// TIA Portal project "学习代码" (V15.1)

(* hardware
DEVICE "S7-1200 station_1"  S7-1200 Station
   slot 0: "Rack_0"  S7-1200 Rack  Rack  V1.0
   slot 1: "PLC_1"  CPU 1214C DC/DC/DC  6ES7 214-1AG40-0XB0  V4.2
   slot 2: "AQ 4x14BIT_1"  6ES7 232-4HD32-0XB0  V2.0
   slot 101: "CM 1241 (RS232)_1"  6ES7 241-1AH32-0XB0  V2.2
*)

// ===== PLC "PLC_1"  CPU 1214C DC/DC/DC =====

VAR_GLOBAL   // PLC tag table "默认变量表"
   "点动模式状态指示灯" AT %Q0.0 : Bool;
   "点动模式标志位" AT %M100.2 : Bool;
   "Last_Status_2" AT %M100.1 : Bool;
   "Last_Status_1" AT %M100.0 : Bool;
   "启动" AT %I1.0 : Bool;
   "停止" AT %I1.1 : Bool;
   "运行标志位" AT %M10.0 : Bool;
   "测试" AT %I1.2 : Bool;
   "测试运行标志位" AT %M10.1 : Bool;
   "传送带运行" AT %Q1.0 : Bool;
   "点动正运行标志位" AT %M10.2 : Bool;
   "点动正" AT %I2.0 : Bool;
   "点动负" AT %I2.1 : Bool;
   "点动负运行标志位" AT %M10.3 : Bool;
   "点动模式选择按钮" AT %I0.0 : Bool;
   "TP输入" AT %I3.0 : Bool;
   "TP输出" AT %Q3.0 : Bool;
   "TON输入" AT %I3.1 : Bool;
   "TON输出" AT %Q3.1 : Bool;
   "TOF输入" AT %I3.2 : Bool;
   "TOF输出" AT %Q3.2 : Bool;
   "TONR输入" AT %I3.3 : Bool;
   "TONR输出" AT %Q3.3 : Bool;
   "TONR复位" AT %I3.4 : Bool;
   "CTU输入" AT %I4.0 : Bool;
   "CTU输出" AT %Q4.0 : Bool;
   "CTD输入" AT %I4.1 : Bool;
   "CTD输出" AT %Q4.1 : Bool;
   "CTUD输入增加" AT %I4.2 : Bool;
   "CTUD输出" AT %Q4.2 : Bool;
   "CTUD输入减少" AT %I4.3 : Bool;
   "比较指令输出" AT %Q4.3 : Bool;
   "数学函数输入" AT %I4.4 : Bool;
   "Clock_1Hz" AT %I4.5 : Bool;
   "Last_Status" AT %M50.0 : Bool;
   "电机1启动信号" AT %I5.0 : Bool;
   "电机1停止信号" AT %I5.1 : Bool;
   "电机1频率加信号" AT %I5.2 : Bool;
   "电机1频率减信号" AT %I5.3 : Bool;
   "电机1运行" AT %Q5.0 : Bool;
   "电机1运行指示灯" AT %Q5.1 : Bool;
   "AQ1" AT %QW96 : Int;
   "System_Byte" AT %MB1 : Byte;
   "FirstScan" AT %M1.0 : Bool;
   "DiagStatusUpdate" AT %M1.1 : Bool;
   "AlwaysTRUE" AT %M1.2 : Bool;
   "AlwaysFALSE" AT %M1.3 : Bool;
END_VAR

TYPE "电机启停运行及速度控制_数据类型"
   STRUCT
      设定运行时间 : Time;
      运行标志 : Bool;
      运行时间到 : Bool;
      频率加信号上次状态 : Bool;
      频率减信号上次状态 : Bool;
      TON_DB : IEC_TIMER;
      给定频率 : Real;
   END_STRUCT;
END_TYPE

DATA_BLOCK "Counter_Data"   // DB1
{ S7_Optimized_Access := 'TRUE' }
VERSION : 0.1
   VAR RETAIN
      CTU : IEC_COUNTER;
   END_VAR
   VAR
      Static_2 : Array[0..1] of IEC_COUNTER;
   END_VAR
BEGIN
END_DATA_BLOCK

DATA_BLOCK "比较指令DB"   // DB2
{ S7_Optimized_Access := 'TRUE' }
VERSION : 0.1
   VAR
      不等于 : Array[0..1] of Int;
      大于 : Real;
      小于 : Time;
      小于等于 : Time_Of_Day;
      大于等于 : DTL;
      INRANGE : Int;
      OUTRANGE : Int;
   END_VAR
BEGIN
END_DATA_BLOCK

DATA_BLOCK "Time_Data"   // DB3
{ S7_Optimized_Access := 'TRUE' }
VERSION : 0.1
   VAR
      TP_DB : IEC_TIMER;
      TON_DB : IEC_TIMER;
      Timer_DB : Array[0..1] of IEC_TIMER;
   END_VAR
BEGIN
END_DATA_BLOCK

DATA_BLOCK "数学函数DB"   // DB4
{ S7_Optimized_Access := 'TRUE' }
VERSION : 0.1
   VAR
      Data1 : Array[0..3] of Int;
      Data2 : Array[0..3] of Int;
      Data3 : Array[0..3] of Real;
      Data4 : Array[0..3] of DInt;
      Data5 : Array[0..1] of DInt;
      Data6 : Array[0..4] of Int;
      Data7 : Array[0..5] of Int;
   END_VAR
BEGIN
END_DATA_BLOCK

DATA_BLOCK "电机启停运行及速度控制_DB"   // DB5
{ S7_Optimized_Access := 'TRUE' }
VERSION : 0.1
   VAR
      电机 : Array[1..4] of "电机启停运行及速度控制_数据类型";
   END_VAR
BEGIN
END_DATA_BLOCK

DATA_BLOCK "电机启停运行及速度控制_FB_DB"   // DB6
{ S7_Optimized_Access := 'TRUE' }
VERSION : 0.1
// stored: InstanceOfName 电机启停运行及速度控制_FB
"电机启停运行及速度控制_FB"
BEGIN
END_DATA_BLOCK

DATA_BLOCK "MODBUS通讯_DB"   // DB7
{ S7_Optimized_Access := 'FALSE' }
VERSION : 0.1
// stored: InstanceOfName MODBUS通讯
"MODBUS通讯"
BEGIN
END_DATA_BLOCK

FUNCTION_BLOCK "Timer_FB"   // FB1, LAD
{ S7_Optimized_Access := 'TRUE' }
VERSION : 0.1
   VAR
      IEC_Timer_0_Instance : TONR_TIME;
   END_VAR
BEGIN

REGION Network 1
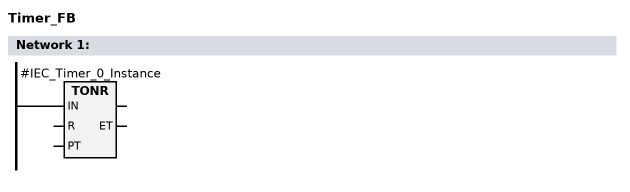
   #IEC_Timer_0_Instance(IN := TRUE);   // TONR
END_REGION
END_FUNCTION_BLOCK

FUNCTION_BLOCK "电机启停运行及速度控制_FB"   // FB2, LAD
{ S7_Optimized_Access := 'TRUE' }
VERSION : 0.1
   VAR_INPUT
      电机启动 : Bool;
      电机停止 : Bool;
      设定运行时间 : Time;
      频率加 : Bool;
      频率减 : Bool;
   END_VAR
   VAR_OUTPUT
      电机输出运行 : Bool;
      运行指示灯 : Bool;
   END_VAR
   VAR_IN_OUT
      给定频率 : Real;
      输出数字量 : Int;
   END_VAR
   VAR
      运行标志 : Bool;
      运行时间到 : Bool;
      IEC_Timer_0_Instance : TON_TIME;
      频率加信号上次状态 : Bool;
      频率减信号上次状态 : Bool;
   END_VAR
   VAR_TEMP
      标定值 : Real;
   END_VAR
   VAR_TEMP   // added for the SCL form of the ladder/FBD networks
      _w1 : Bool;
   END_VAR
BEGIN

REGION Network 1: 启动
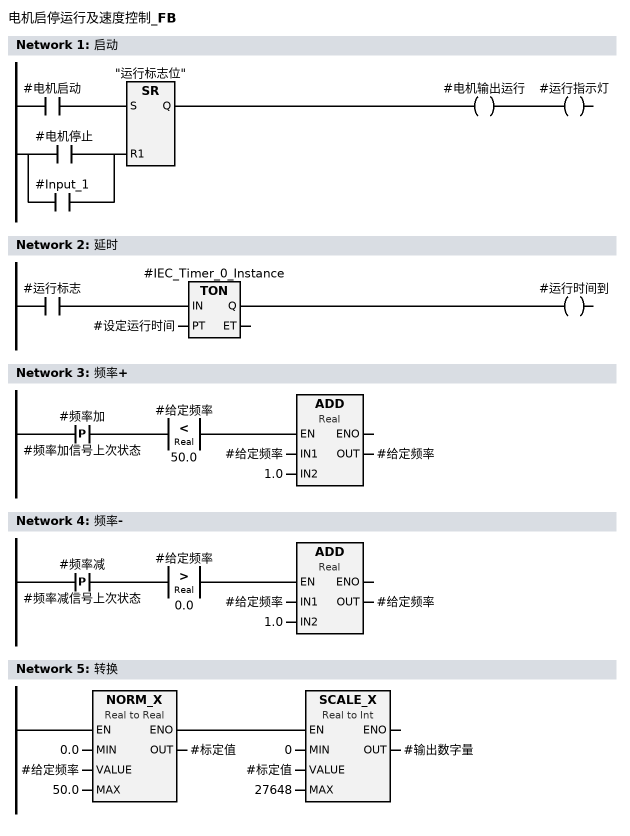
   RUNG wire#powerrail
      Contact( #电机启动 )
      S_SR(operand := "运行标志位", r1 := wire#w1)
      Coil( #电机输出运行 )
      Coil( #运行指示灯 )
   END_RUNG
   RUNG wire#powerrail
      Contact( #电机停止 )
   END_RUNG wire#w1
   RUNG wire#powerrail
      Contact( #Input_1 )
   END_RUNG wire#w1
   // the same network as SCL:
   IF #电机启动 THEN
       "运行标志位" := TRUE;   // SR flip-flop
   END_IF;
   IF #电机停止 OR #Input_1 THEN "运行标志位" := FALSE; END_IF;
   #电机输出运行 := "运行标志位";
   #运行指示灯 := "运行标志位";
END_REGION

REGION Network 2: 延时
   #IEC_Timer_0_Instance(IN := #运行标志, PT := #设定运行时间);   // TON
   #运行时间到 := #IEC_Timer_0_Instance.Q;
END_REGION

REGION Network 3: 频率+
   RUNG wire#powerrail
      P_Contact(operand := #频率加, bit := #频率加信号上次状态)
      { S7_Templates := "SrcType := Real" } LT_Contact(in1 := #给定频率, in2 := 50.0)
      { S7_Templates := "SrcType := Real"; S7_GenerateENO := "TRUE" } Add(in1 := #给定频率, in2 := 1.0, out => #给定频率)
   END_RUNG
   // the same network as SCL:
   #_w1 := #频率加 AND NOT #频率加信号上次状态;   // rising edge of #频率加
   #频率加信号上次状态 := #频率加;
   IF #_w1 AND (#给定频率 < 50.0) THEN #给定频率 := #给定频率 + 1.0; END_IF;
END_REGION

REGION Network 4: 频率-
   RUNG wire#powerrail
      P_Contact(operand := #频率减, bit := #频率减信号上次状态)
      { S7_Templates := "SrcType := Real" } GT_Contact(in1 := #给定频率, in2 := 0.0)
      { S7_Templates := "SrcType := Real"; S7_GenerateENO := "TRUE" } Add(in1 := #给定频率, in2 := 1.0, out => #给定频率)
   END_RUNG
   // the same network as SCL:
   #_w1 := #频率减 AND NOT #频率减信号上次状态;   // rising edge of #频率减
   #频率减信号上次状态 := #频率减;
   IF #_w1 AND (#给定频率 > 0.0) THEN #给定频率 := #给定频率 + 1.0; END_IF;
END_REGION

REGION Network 5: 转换
   RUNG wire#powerrail
      { S7_Templates := "[SrcType := Real, DestType := Real]"; S7_GenerateENO := "TRUE" } Normalize(min := 0.0, value := #给定频率, max := 50.0, out => #标定值)
      { S7_Templates := "[SrcType := Real, DestType := Int]"; S7_GenerateENO := "TRUE" } Scale(min := 0, value := #标定值, max := 27648, out => #输出数字量)
   END_RUNG
   // the same network as SCL:
   // ENO of a box is taken as its EN; it also drops when the box reports an error
   #标定值 := NORM_X(MIN := 0.0, VALUE := #给定频率, MAX := 50.0);
   #输出数字量 := SCALE_X(MIN := 0, VALUE := #标定值, MAX := 27648);
END_REGION
END_FUNCTION_BLOCK

FUNCTION_BLOCK "MODBUS通讯"   // FB3, LAD
{ S7_Optimized_Access := 'FALSE' }
VERSION : 0.1
   VAR_INPUT
      初始化 : Bool;
      正转 : Bool;
      反转 : Bool;
      停止 : Bool;
      频率设定 : Real;
   END_VAR
   VAR_OUTPUT
      输出频率 : Real;
      输出电流 : Real;
      输出电压 : Real;
   END_VAR
   VAR
      Modbus_Comm_Load_DB : Modbus_Comm_Load;
      MB_Com_load : Struct
         Done : Bool;
         Error : Bool;
         Status : Word;
      END_STRUCT;
      MB_Mast_step : USInt;
      Modbus_Master_DB : Modbus_Master;
      MD_Master_write : Struct
         Data_ptr : Array[0..1] of Int;
         Done : Bool;
         Busy : Bool;
         Error : Bool;
         Status : Word;
      END_STRUCT;
      MD_Master_status : Struct
         Data_ptr : Array[0..0] of Int;
         Done : Bool;
         Busy : Bool;
         Error : Bool;
         Status : Word;
      END_STRUCT;
      MD_Master_RD : Struct
         Data_ptr : Array[0..3] of Int;
         Done : Bool;
         Busy : Bool;
         Error : Bool;
         Status : Word;
      END_STRUCT;
   END_VAR
   VAR_TEMP
      设定频率_Real : Real;
      输出频率_Real : Real;
      输出电流_Real : Real;
      输出电压_Real : Real;
   END_VAR
BEGIN

REGION Network 1
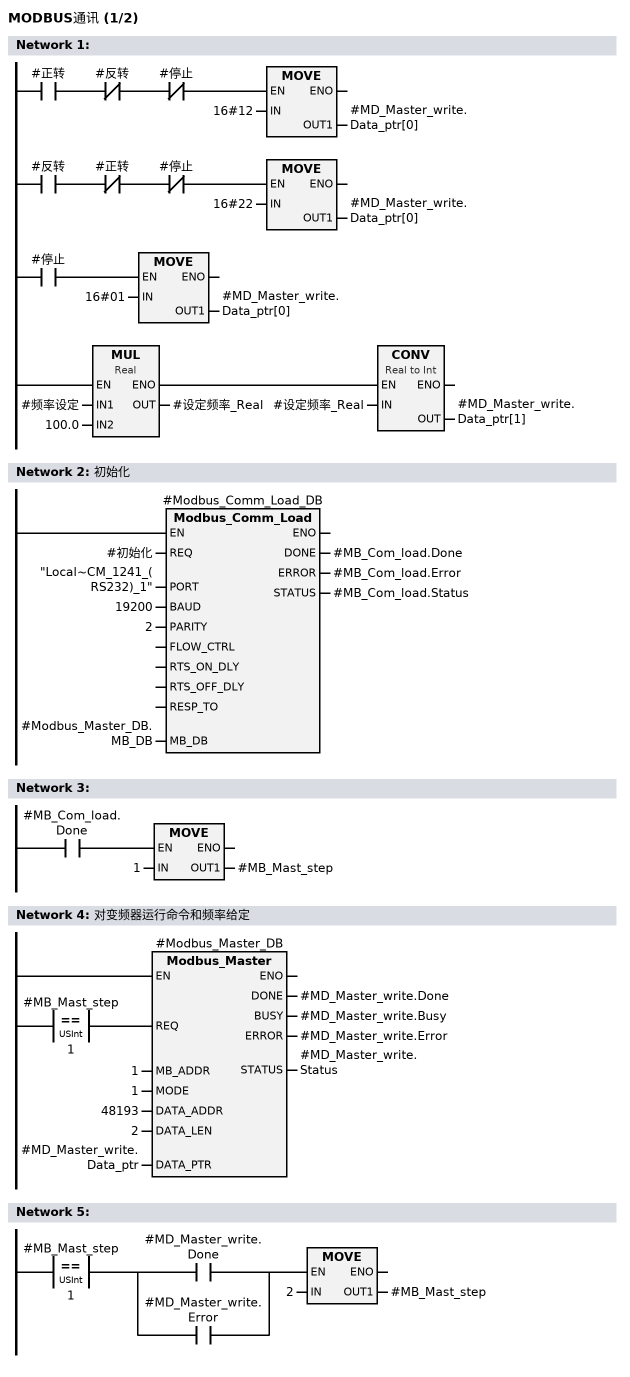
   RUNG wire#powerrail
      Contact( #正转 )
      I_Contact( #反转 )
      I_Contact( #停止 )
      { S7_GenerateENO := "TRUE" } Move(in := 16#12, out1 => #MD_Master_write.Data_ptr[0])
   END_RUNG
   RUNG wire#powerrail
      Contact( #反转 )
      I_Contact( #正转 )
      I_Contact( #停止 )
      { S7_GenerateENO := "TRUE" } Move(in := 16#22, out1 => #MD_Master_write.Data_ptr[0])
   END_RUNG
   RUNG wire#powerrail
      Contact( #停止 )
      { S7_GenerateENO := "TRUE" } Move(in := 16#01, out1 => #MD_Master_write.Data_ptr[0])
   END_RUNG
   RUNG wire#powerrail
      { S7_Templates := "SrcType := Real"; S7_GenerateENO := "TRUE" } Mul(in1 := #频率设定, in2 := 100.0, out => #设定频率_Real)
      { S7_Templates := "[SrcType := Real, DestType := Int]"; S7_GenerateENO := "TRUE" } Convert(in := #设定频率_Real, out => #MD_Master_write.Data_ptr[1])
   END_RUNG
   RUNG wire#powerrail
   END_RUNG
   // the same network as SCL:
   // ENO of a box is taken as its EN; it also drops when the box reports an error
   IF #正转 AND NOT #反转 AND NOT #停止 THEN #MD_Master_write.Data_ptr[0] := 16#12; END_IF;
   IF #反转 AND NOT #正转 AND NOT #停止 THEN #MD_Master_write.Data_ptr[0] := 16#22; END_IF;
   IF #停止 THEN #MD_Master_write.Data_ptr[0] := 16#01; END_IF;
   #设定频率_Real := #频率设定 * 100.0;
   #MD_Master_write.Data_ptr[1] := REAL_TO_INT(#设定频率_Real);
END_REGION

REGION Network 2: 初始化
   #Modbus_Comm_Load_DB(REQ := #初始化,   // Modbus_Comm_Load
                        PORT := "Local~CM_1241_(RS232)_1",
                        BAUD := 19200,
                        PARITY := 2,
                        MB_DB := #Modbus_Master_DB.MB_DB,
                        DONE => #MB_Com_load.Done,
                        ERROR => #MB_Com_load.Error,
                        STATUS => #MB_Com_load.Status);
END_REGION

REGION Network 3
   RUNG wire#powerrail
      Contact( #MB_Com_load.Done )
      { S7_GenerateENO := "TRUE" } Move(in := 1, out1 => #MB_Mast_step)
   END_RUNG
   // the same network as SCL:
   IF #MB_Com_load.Done THEN #MB_Mast_step := 1; END_IF;
END_REGION

REGION Network 4: 对变频器运行命令和频率给定
   #Modbus_Master_DB(REQ := #MB_Mast_step = 1,   // Modbus_Master
                     MB_ADDR := 1,
                     MODE := 1,
                     DATA_ADDR := 48193,
                     DATA_LEN := 2,
                     DATA_PTR := #MD_Master_write.Data_ptr,
                     DONE => #MD_Master_write.Done,
                     BUSY => #MD_Master_write.Busy,
                     ERROR => #MD_Master_write.Error,
                     STATUS => #MD_Master_write.Status);
END_REGION

REGION Network 5
   RUNG wire#powerrail
      { S7_Templates := "SrcType := USInt" } EQ_Contact(in1 := #MB_Mast_step, in2 := 1)
      wire#w1
      Contact( #MD_Master_write.Done )
      wire#w2
      { S7_GenerateENO := "TRUE" } Move(in := 2, out1 => #MB_Mast_step)
   END_RUNG
   RUNG wire#w1
      Contact( #MD_Master_write.Error )
   END_RUNG wire#w2
   // the same network as SCL:
   IF (#MB_Mast_step = 1) AND (#MD_Master_write.Done OR #MD_Master_write.Error) THEN
       #MB_Mast_step := 2;
   END_IF;
END_REGION

REGION Network 6: 读变频器状态
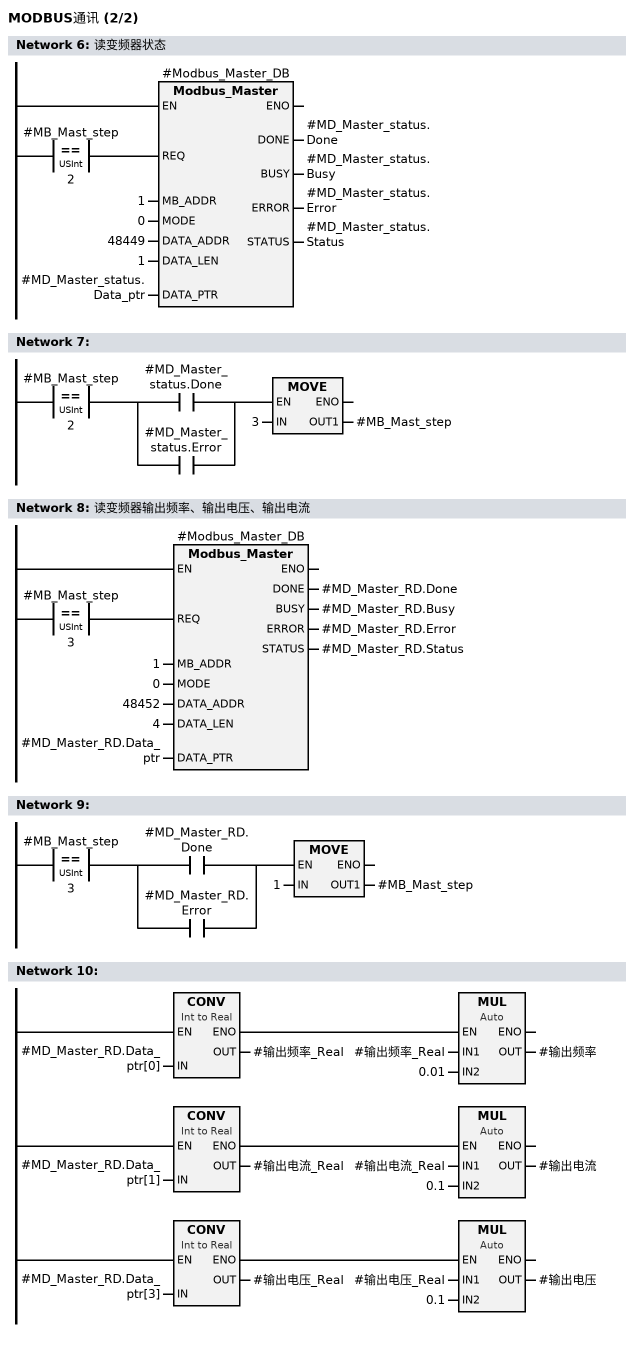
   #Modbus_Master_DB(REQ := #MB_Mast_step = 2,   // Modbus_Master
                     MB_ADDR := 1,
                     MODE := 0,
                     DATA_ADDR := 48449,
                     DATA_LEN := 1,
                     DATA_PTR := #MD_Master_status.Data_ptr,
                     DONE => #MD_Master_status.Done,
                     BUSY => #MD_Master_status.Busy,
                     ERROR => #MD_Master_status.Error,
                     STATUS => #MD_Master_status.Status);
END_REGION

REGION Network 7
   RUNG wire#powerrail
      { S7_Templates := "SrcType := USInt" } EQ_Contact(in1 := #MB_Mast_step, in2 := 2)
      wire#w1
      Contact( #MD_Master_status.Done )
      wire#w2
      { S7_GenerateENO := "TRUE" } Move(in := 3, out1 => #MB_Mast_step)
   END_RUNG
   RUNG wire#w1
      Contact( #MD_Master_status.Error )
   END_RUNG wire#w2
   // the same network as SCL:
   IF (#MB_Mast_step = 2) AND (#MD_Master_status.Done OR #MD_Master_status.Error) THEN
       #MB_Mast_step := 3;
   END_IF;
END_REGION

REGION Network 8: 读变频器输出频率、输出电压、输出电流
   #Modbus_Master_DB(REQ := #MB_Mast_step = 3,   // Modbus_Master
                     MB_ADDR := 1,
                     MODE := 0,
                     DATA_ADDR := 48452,
                     DATA_LEN := 4,
                     DATA_PTR := #MD_Master_RD.Data_ptr,
                     DONE => #MD_Master_RD.Done,
                     BUSY => #MD_Master_RD.Busy,
                     ERROR => #MD_Master_RD.Error,
                     STATUS => #MD_Master_RD.Status);
END_REGION

REGION Network 9
   RUNG wire#powerrail
      { S7_Templates := "SrcType := USInt" } EQ_Contact(in1 := #MB_Mast_step, in2 := 3)
      wire#w1
      Contact( #MD_Master_RD.Done )
      wire#w2
      { S7_GenerateENO := "TRUE" } Move(in := 1, out1 => #MB_Mast_step)
   END_RUNG
   RUNG wire#w1
      Contact( #MD_Master_RD.Error )
   END_RUNG wire#w2
   // the same network as SCL:
   IF (#MB_Mast_step = 3) AND (#MD_Master_RD.Done OR #MD_Master_RD.Error) THEN #MB_Mast_step := 1; END_IF;
END_REGION

REGION Network 10
   RUNG wire#powerrail
      { S7_Templates := "[SrcType := Int, DestType := Real]"; S7_GenerateENO := "TRUE" } Convert(in := #MD_Master_RD.Data_ptr[0], out => #输出频率_Real)
      { S7_GenerateENO := "TRUE" } Mul(in1 := #输出频率_Real, in2 := 0.01, out => #输出频率)
   END_RUNG
   RUNG wire#powerrail
      { S7_Templates := "[SrcType := Int, DestType := Real]"; S7_GenerateENO := "TRUE" } Convert(in := #MD_Master_RD.Data_ptr[1], out => #输出电流_Real)
      { S7_GenerateENO := "TRUE" } Mul(in1 := #输出电流_Real, in2 := 0.1, out => #输出电流)
   END_RUNG
   RUNG wire#powerrail
      { S7_Templates := "[SrcType := Int, DestType := Real]"; S7_GenerateENO := "TRUE" } Convert(in := #MD_Master_RD.Data_ptr[3], out => #输出电压_Real)
      { S7_GenerateENO := "TRUE" } Mul(in1 := #输出电压_Real, in2 := 0.1, out => #输出电压)
   END_RUNG
   // the same network as SCL:
   // ENO of a box is taken as its EN; it also drops when the box reports an error
   #输出频率_Real := INT_TO_REAL(#MD_Master_RD.Data_ptr[0]);
   #输出频率 := #输出频率_Real * 0.01;
   #输出电流_Real := INT_TO_REAL(#MD_Master_RD.Data_ptr[1]);
   #输出电流 := #输出电流_Real * 0.1;
   #输出电压_Real := INT_TO_REAL(#MD_Master_RD.Data_ptr[3]);
   #输出电压 := #输出电压_Real * 0.1;
END_REGION
END_FUNCTION_BLOCK

FUNCTION "传送带控制" : Void   // FC1, LAD
{ S7_Optimized_Access := 'TRUE' }
VERSION : 0.1
   VAR_TEMP   // added for the SCL form of the ladder/FBD networks
      _w1 : Bool;
      _w2 : Bool;
   END_VAR
BEGIN

REGION Network 1
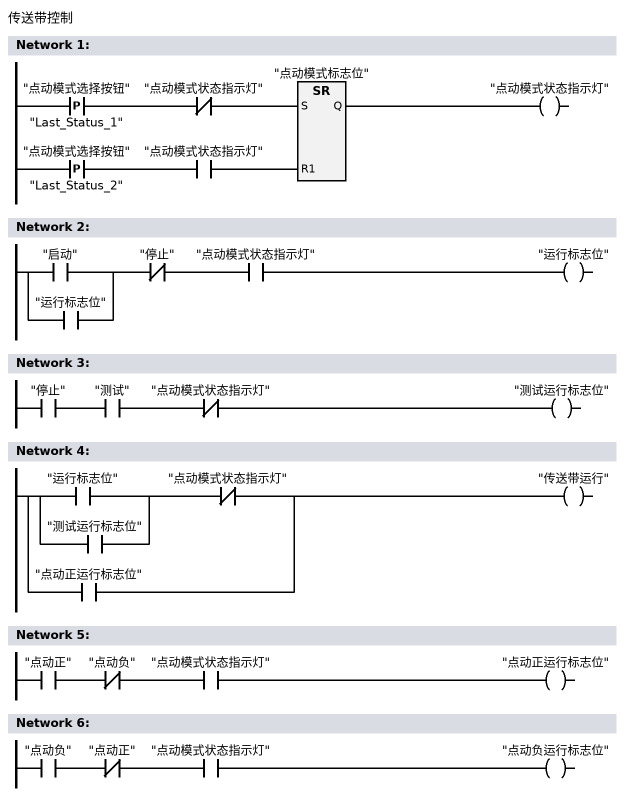
   RUNG wire#powerrail
      P_Contact(operand := "点动模式选择按钮", bit := "Last_Status_1")
      I_Contact( "点动模式状态指示灯" )
      S_SR(operand := "点动模式标志位", r1 := wire#w1)
      Coil( "点动模式状态指示灯" )
   END_RUNG
   RUNG wire#powerrail
      P_Contact(operand := "点动模式选择按钮", bit := "Last_Status_2")
      Contact( "点动模式状态指示灯" )
   END_RUNG wire#w1
   // the same network as SCL:
   #_w1 := "点动模式选择按钮" AND NOT "Last_Status_1";   // rising edge of "点动模式选择按钮"
   "Last_Status_1" := "点动模式选择按钮";
   #_w2 := "点动模式选择按钮" AND NOT "Last_Status_2";   // rising edge of "点动模式选择按钮"
   "Last_Status_2" := "点动模式选择按钮";
   IF #_w1 AND NOT "点动模式状态指示灯" THEN
       "点动模式标志位" := TRUE;   // SR flip-flop
   END_IF;
   IF #_w2 AND "点动模式状态指示灯" THEN "点动模式标志位" := FALSE; END_IF;
   "点动模式状态指示灯" := "点动模式标志位";
END_REGION

REGION Network 2
   RUNG wire#powerrail
      Contact( "启动" )
      wire#w1
      I_Contact( "停止" )
      Contact( "点动模式状态指示灯" )
      Coil( "运行标志位" )
   END_RUNG
   RUNG wire#powerrail
      Contact( "运行标志位" )
   END_RUNG wire#w1
   // the same network as SCL:
   "运行标志位" := ("启动" OR "运行标志位") AND NOT "停止" AND "点动模式状态指示灯";
END_REGION

REGION Network 3
   RUNG wire#powerrail
      Contact( "停止" )
      Contact( "测试" )
      I_Contact( "点动模式状态指示灯" )
      Coil( "测试运行标志位" )
   END_RUNG
   // the same network as SCL:
   "测试运行标志位" := "停止" AND "测试" AND NOT "点动模式状态指示灯";
END_REGION

REGION Network 4
   RUNG wire#powerrail
      Contact( "运行标志位" )
      wire#w1
      I_Contact( "点动模式状态指示灯" )
      wire#w2
      Coil( "传送带运行" )
   END_RUNG
   RUNG wire#powerrail
      Contact( "测试运行标志位" )
   END_RUNG wire#w1
   RUNG wire#powerrail
      Contact( "点动正运行标志位" )
   END_RUNG wire#w2
   // the same network as SCL:
   "传送带运行" := (("运行标志位" OR "测试运行标志位") AND NOT "点动模式状态指示灯") OR "点动正运行标志位";
END_REGION

REGION Network 5
   RUNG wire#powerrail
      Contact( "点动正" )
      I_Contact( "点动负" )
      Contact( "点动模式状态指示灯" )
      Coil( "点动正运行标志位" )
   END_RUNG
   // the same network as SCL:
   "点动正运行标志位" := "点动正" AND NOT "点动负" AND "点动模式状态指示灯";
END_REGION

REGION Network 6
   RUNG wire#powerrail
      Contact( "点动负" )
      I_Contact( "点动正" )
      Contact( "点动模式状态指示灯" )
      Coil( "点动负运行标志位" )
   END_RUNG
   // the same network as SCL:
   "点动负运行标志位" := "点动负" AND NOT "点动正" AND "点动模式状态指示灯";
END_REGION
END_FUNCTION

FUNCTION "Timer" : Void   // FC2, LAD
{ S7_Optimized_Access := 'TRUE' }
VERSION : 0.1
BEGIN

REGION Network 1
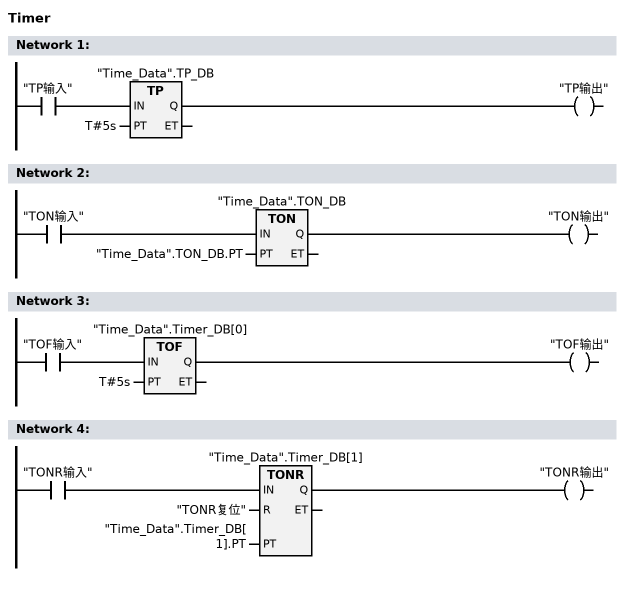
   "Time_Data".TP_DB.TP(IN := "TP输入", PT := T#5s);
   "TP输出" := "Time_Data".TP_DB.Q;
END_REGION

REGION Network 2
   "Time_Data".TON_DB.TON(IN := "TON输入", PT := "Time_Data".TON_DB.PT);
   "TON输出" := "Time_Data".TON_DB.Q;
END_REGION

REGION Network 3
   "Time_Data".Timer_DB[0].TOF(IN := "TOF输入", PT := T#5s);
   "TOF输出" := "Time_Data".Timer_DB[0].Q;
END_REGION

REGION Network 4
   "Time_Data".Timer_DB[1].TONR(IN := "TONR输入", R := "TONR复位", PT := "Time_Data".Timer_DB[1].PT);
   "TONR输出" := "Time_Data".Timer_DB[1].Q;
END_REGION
END_FUNCTION

FUNCTION "Counter" : Void   // FC3, LAD
{ S7_Optimized_Access := 'TRUE' }
VERSION : 0.1
BEGIN

REGION Network 1
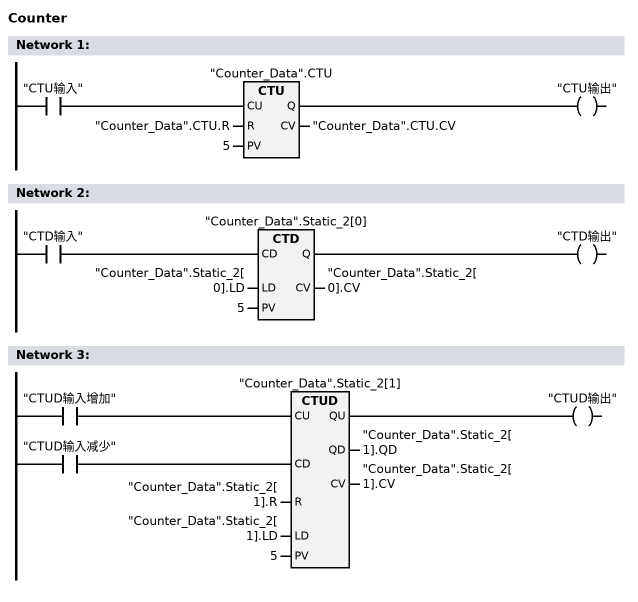
   "Counter_Data".CTU.CTU(CU := "CTU输入", R := "Counter_Data".CTU.R, PV := 5, CV => "Counter_Data".CTU.CV);
   "CTU输出" := "Counter_Data".CTU.Q;
END_REGION

REGION Network 2
   "Counter_Data".Static_2[0].CTD(CD := "CTD输入",
                           LD := "Counter_Data".Static_2[0].LD,
                           PV := 5,
                           CV => "Counter_Data".Static_2[0].CV);
   "CTD输出" := "Counter_Data".Static_2[0].Q;
END_REGION

REGION Network 3
   "Counter_Data".Static_2[1].CTUD(CU := "CTUD输入增加",
                           CD := "CTUD输入减少",
                           R := "Counter_Data".Static_2[1].R,
                           LD := "Counter_Data".Static_2[1].LD,
                           PV := 5,
                           QD => "Counter_Data".Static_2[1].QD,
                           CV => "Counter_Data".Static_2[1].CV);
   "CTUD输出" := "Counter_Data".Static_2[1].QU;
END_REGION
END_FUNCTION

FUNCTION "比较指令" : Void   // FC4, LAD
{ S7_Optimized_Access := 'TRUE' }
VERSION : 0.1
BEGIN

REGION Network 1
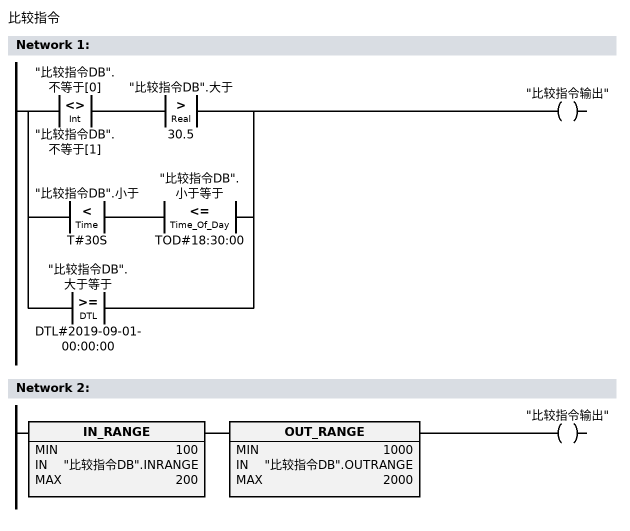
   RUNG wire#powerrail
      { S7_Templates := "SrcType := Int" } NE_Contact(in1 := "比较指令DB".不等于[0], in2 := "比较指令DB".不等于[1])
      { S7_Templates := "SrcType := Real" } GT_Contact(in1 := "比较指令DB".大于, in2 := 30.5)
      wire#w1
      Coil( "比较指令输出" )
   END_RUNG
   RUNG wire#powerrail
      { S7_Templates := "SrcType := Time" } LT_Contact(in1 := "比较指令DB".小于, in2 := T#30S)
      { S7_Templates := "SrcType := Time_Of_Day" } LE_Contact(in1 := "比较指令DB".小于等于, in2 := TOD#18:30:00)
   END_RUNG wire#w1
   RUNG wire#powerrail
      { S7_Templates := "SrcType := DTL" } GE_Contact(in1 := "比较指令DB".大于等于, in2 := DTL#2019-09-01-00:00:00)
   END_RUNG wire#w1
   // the same network as SCL:
   "比较指令输出" := (("比较指令DB".不等于[0] <> "比较指令DB".不等于[1]) AND ("比较指令DB".大于 > 30.5)) OR (("比较指令DB".小于 < T#30S) AND ("比较指令DB".小于等于 <= TOD#18:30:00)) OR ("比较指令DB".大于等于 >= DTL#2019-09-01-00:00:00);
END_REGION

REGION Network 2
   "比较指令输出" := (100 <= "比较指令DB".INRANGE) AND ("比较指令DB".INRANGE <= 200) AND (("比较指令DB".OUTRANGE < 1000) OR ("比较指令DB".OUTRANGE > 2000));
END_REGION
END_FUNCTION

FUNCTION "数学函数" : Void   // FC5, LAD
{ S7_Optimized_Access := 'TRUE' }
VERSION : 0.1
   VAR_INPUT
      "M10.0" : Bool;
   END_VAR
   VAR_TEMP   // added for the SCL form of the ladder/FBD networks
      _w1 : Bool;
   END_VAR
BEGIN

REGION Network 1
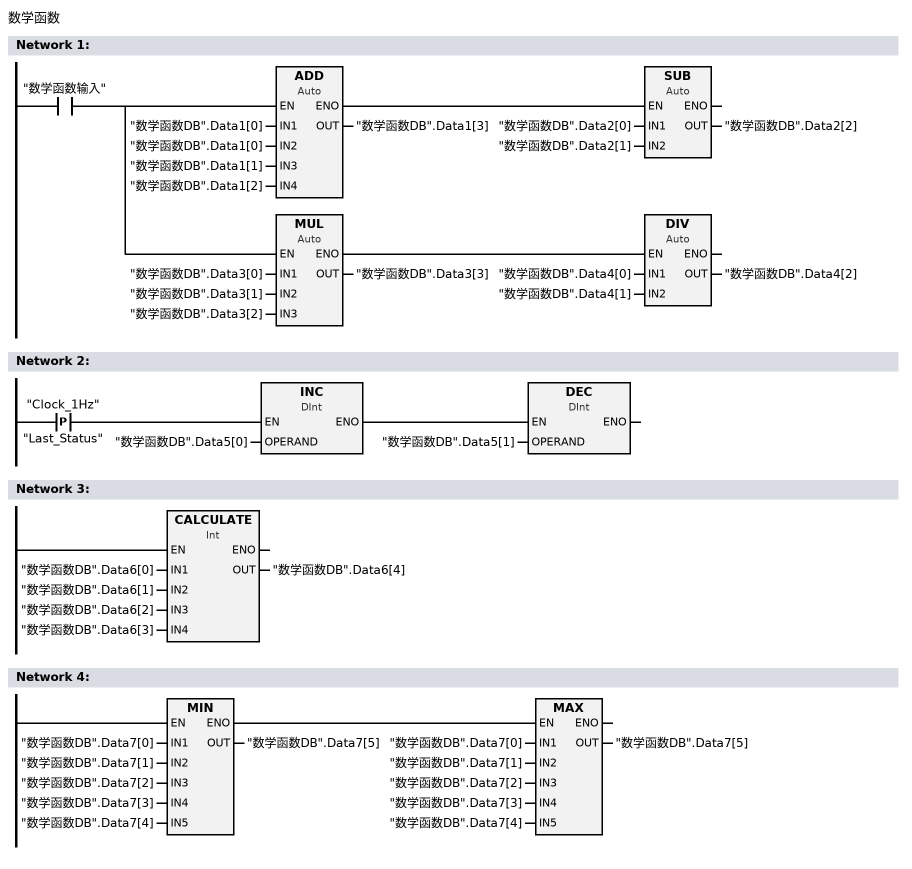
   RUNG wire#powerrail
      Contact( "数学函数输入" )
      wire#w1
      Add(in1 := "数学函数DB".Data1[0], in2 := "数学函数DB".Data1[0], in3 := "数学函数DB".Data1[1], in4 := "数学函数DB".Data1[2], out => "数学函数DB".Data1[3])
      Sub(in1 := "数学函数DB".Data2[0], in2 := "数学函数DB".Data2[1], out => "数学函数DB".Data2[2])
   END_RUNG
   RUNG wire#w1
      Mul(in1 := "数学函数DB".Data3[0], in2 := "数学函数DB".Data3[1], in3 := "数学函数DB".Data3[2], out => "数学函数DB".Data3[3])
      { S7_GenerateENO := "TRUE" } Div(in1 := "数学函数DB".Data4[0], in2 := "数学函数DB".Data4[1], out => "数学函数DB".Data4[2])
   END_RUNG
   // the same network as SCL:
   IF "数学函数输入" THEN
       "数学函数DB".Data1[3] := "数学函数DB".Data1[0] + "数学函数DB".Data1[0] + "数学函数DB".Data1[1] + "数学函数DB".Data1[2];
       "数学函数DB".Data2[2] := "数学函数DB".Data2[0] - "数学函数DB".Data2[1];
       "数学函数DB".Data3[3] := "数学函数DB".Data3[0] * "数学函数DB".Data3[1] * "数学函数DB".Data3[2];
       "数学函数DB".Data4[2] := "数学函数DB".Data4[0] / "数学函数DB".Data4[1];
   END_IF;
END_REGION

REGION Network 2
   RUNG wire#powerrail
      P_Contact(operand := "Clock_1Hz", bit := "Last_Status")
      { S7_Templates := "DestType := DInt"; S7_GenerateENO := "TRUE" } Inc( "数学函数DB".Data5[0] )
      { S7_Templates := "DestType := DInt"; S7_GenerateENO := "TRUE" } Dec( "数学函数DB".Data5[1] )
   END_RUNG
   // the same network as SCL:
   // ENO of a box is taken as its EN; it also drops when the box reports an error
   #_w1 := "Clock_1Hz" AND NOT "Last_Status";   // rising edge of "Clock_1Hz"
   "Last_Status" := "Clock_1Hz";
   IF #_w1 THEN
       "数学函数DB".Data5[0] := "数学函数DB".Data5[0] + 1;
       "数学函数DB".Data5[1] := "数学函数DB".Data5[1] - 1;
   END_IF;
END_REGION

REGION Network 3
   RUNG wire#powerrail
      { S7_Templates := "SrcType := Int"; S7_GenerateENO := "TRUE"; S7_Expression := "(IN1 + IN2) * (IN1 - IN2) - (IN3 + IN4) * (IN3 - IN4)" } Calculate(in1 := "数学函数DB".Data6[0], in2 := "数学函数DB".Data6[1], in3 := "数学函数DB".Data6[2], in4 := "数学函数DB".Data6[3], out => "数学函数DB".Data6[4])
   END_RUNG
   // the same network as SCL:
   "数学函数DB".Data6[4] := ("数学函数DB".Data6[0] + "数学函数DB".Data6[1]) * ("数学函数DB".Data6[0] - "数学函数DB".Data6[1]) - ("数学函数DB".Data6[2] + "数学函数DB".Data6[3]) * ("数学函数DB".Data6[2] - "数学函数DB".Data6[3]);
END_REGION

REGION Network 4
   // ENO of a box is taken as its EN; it also drops when the box reports an error
   "数学函数DB".Data7[5] := MIN(IN1 := "数学函数DB".Data7[0], IN2 := "数学函数DB".Data7[1], IN3 := "数学函数DB".Data7[2], IN4 := "数学函数DB".Data7[3], IN5 := "数学函数DB".Data7[4]);
   "数学函数DB".Data7[5] := MAX(IN1 := "数学函数DB".Data7[0], IN2 := "数学函数DB".Data7[1], IN3 := "数学函数DB".Data7[2], IN4 := "数学函数DB".Data7[3], IN5 := "数学函数DB".Data7[4]);
END_REGION
END_FUNCTION

FUNCTION "电机启停运行及速度控制" : Void   // FC6, LAD
{ S7_Optimized_Access := 'TRUE' }
VERSION : 0.1
   VAR_INPUT
      电机启动 : Bool;
      电机停止 : Bool;
      设定运行时间 : Time;
      频率加 : Bool;
      频率减 : Bool;
   END_VAR
   VAR_OUTPUT
      电机输出运行 : Bool;
      运行指示灯 : Bool;
      输出数字量 : Int;
   END_VAR
   VAR_IN_OUT
      运行标志 : Bool;
      运行时间到 : Bool;
      TON_DB : IEC_TIMER;
      频率加信号上次状态 : Bool;
      频率减信号上次状态 : Bool;
      给定频率 : Real;
   END_VAR
   VAR_TEMP
      标定值 : Real;
   END_VAR
   VAR_TEMP   // added for the SCL form of the ladder/FBD networks
      _w1 : Bool;
   END_VAR
BEGIN

REGION Network 1: 启动
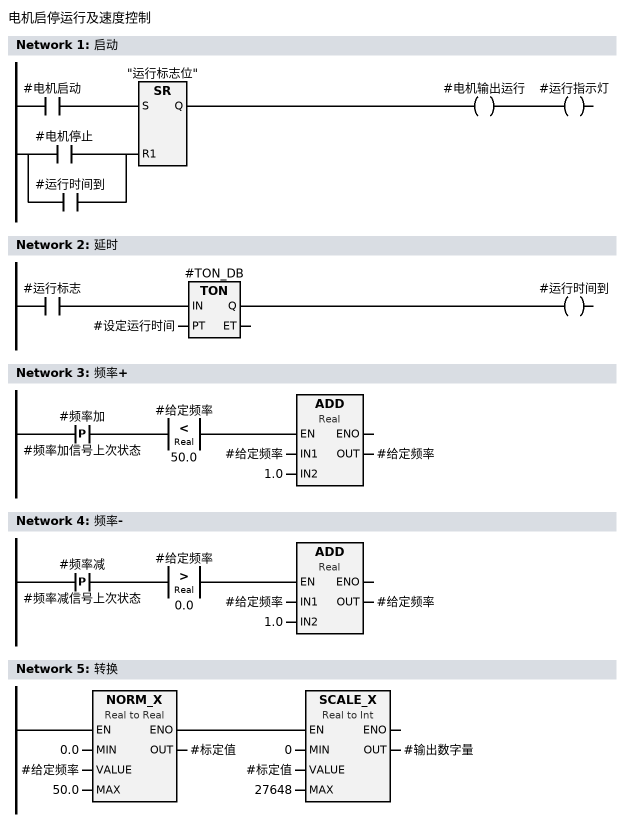
   RUNG wire#powerrail
      Contact( #电机启动 )
      S_SR(operand := "运行标志位", r1 := wire#w1)
      Coil( #电机输出运行 )
      Coil( #运行指示灯 )
   END_RUNG
   RUNG wire#powerrail
      Contact( #电机停止 )
   END_RUNG wire#w1
   RUNG wire#powerrail
      Contact( #运行时间到 )
   END_RUNG wire#w1
   // the same network as SCL:
   IF #电机启动 THEN
       "运行标志位" := TRUE;   // SR flip-flop
   END_IF;
   IF #电机停止 OR #运行时间到 THEN "运行标志位" := FALSE; END_IF;
   #电机输出运行 := "运行标志位";
   #运行指示灯 := "运行标志位";
END_REGION

REGION Network 2: 延时
   #TON_DB.TON(IN := #运行标志, PT := #设定运行时间);
   #运行时间到 := #TON_DB.Q;
END_REGION

REGION Network 3: 频率+
   RUNG wire#powerrail
      P_Contact(operand := #频率加, bit := #频率加信号上次状态)
      { S7_Templates := "SrcType := Real" } LT_Contact(in1 := #给定频率, in2 := 50.0)
      { S7_Templates := "SrcType := Real"; S7_GenerateENO := "TRUE" } Add(in1 := #给定频率, in2 := 1.0, out => #给定频率)
   END_RUNG
   // the same network as SCL:
   #_w1 := #频率加 AND NOT #频率加信号上次状态;   // rising edge of #频率加
   #频率加信号上次状态 := #频率加;
   IF #_w1 AND (#给定频率 < 50.0) THEN #给定频率 := #给定频率 + 1.0; END_IF;
END_REGION

REGION Network 4: 频率-
   RUNG wire#powerrail
      P_Contact(operand := #频率减, bit := #频率减信号上次状态)
      { S7_Templates := "SrcType := Real" } GT_Contact(in1 := #给定频率, in2 := 0.0)
      { S7_Templates := "SrcType := Real"; S7_GenerateENO := "TRUE" } Add(in1 := #给定频率, in2 := 1.0, out => #给定频率)
   END_RUNG
   // the same network as SCL:
   #_w1 := #频率减 AND NOT #频率减信号上次状态;   // rising edge of #频率减
   #频率减信号上次状态 := #频率减;
   IF #_w1 AND (#给定频率 > 0.0) THEN #给定频率 := #给定频率 + 1.0; END_IF;
END_REGION

REGION Network 5: 转换
   RUNG wire#powerrail
      { S7_Templates := "[SrcType := Real, DestType := Real]"; S7_GenerateENO := "TRUE" } Normalize(min := 0.0, value := #给定频率, max := 50.0, out => #标定值)
      { S7_Templates := "[SrcType := Real, DestType := Int]"; S7_GenerateENO := "TRUE" } Scale(min := 0, value := #标定值, max := 27648, out => #输出数字量)
   END_RUNG
   // the same network as SCL:
   // ENO of a box is taken as its EN; it also drops when the box reports an error
   #标定值 := NORM_X(MIN := 0.0, VALUE := #给定频率, MAX := 50.0);
   #输出数字量 := SCALE_X(MIN := 0, VALUE := #标定值, MAX := 27648);
END_REGION
END_FUNCTION

ORGANIZATION_BLOCK "Main"   // OB1, LAD, ProgramCycle
TITLE = "Main Program Sweep (Cycle)"
{ S7_Optimized_Access := 'TRUE' }
VERSION : 0.1
   VAR_INPUT
      Initial_Call : Bool;   // Initial call of this OB
      Remanence : Bool;   // =True, if remanent data are available
   END_VAR
BEGIN

REGION Network 1
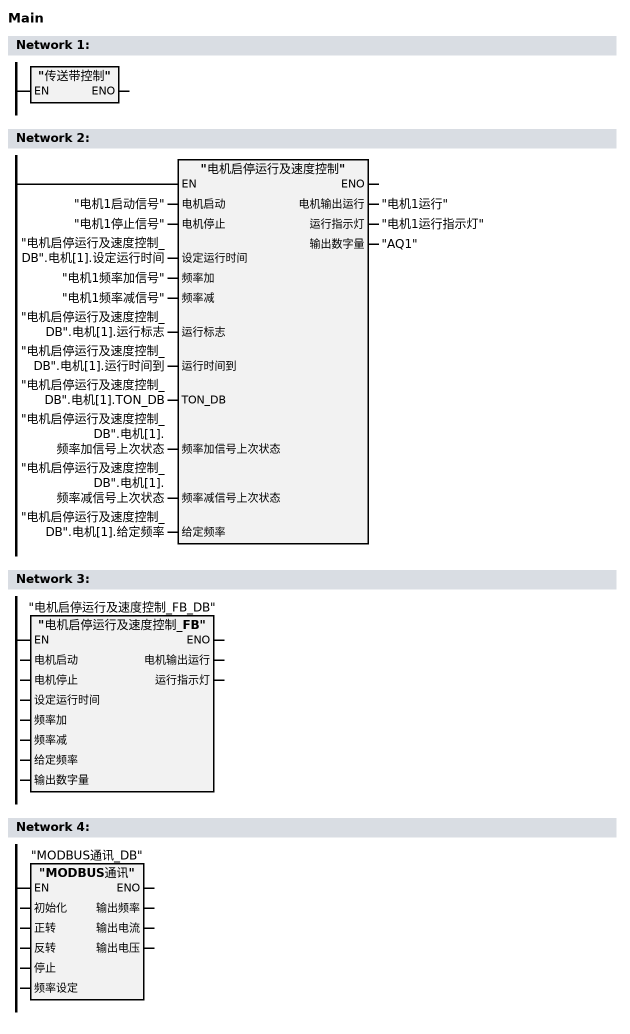
   RUNG wire#powerrail
      "传送带控制"()
   END_RUNG
   // the same network as SCL:
   "传送带控制"();
END_REGION

REGION Network 2
   RUNG wire#powerrail
      "电机启停运行及速度控制"(电机启动 := "电机1启动信号", 电机停止 := "电机1停止信号", 设定运行时间 := "电机启停运行及速度控制_DB".电机[1].设定运行时间, 频率加 := "电机1频率加信号", 频率减 := "电机1频率减信号", 运行标志 := "电机启停运行及速度控制_DB".电机[1].运行标志, 运行时间到 := "电机启停运行及速度控制_DB".电机[1].运行时间到, TON_DB := "电机启停运行及速度控制_DB".电机[1].TON_DB, 频率加信号上次状态 := "电机启停运行及速度控制_DB".电机[1].频率加信号上次状态, 频率减信号上次状态 := "电机启停运行及速度控制_DB".电机[1].频率减信号上次状态, 给定频率 := "电机启停运行及速度控制_DB".电机[1].给定频率, 电机输出运行 => "电机1运行", 运行指示灯 => "电机1运行指示灯", 输出数字量 => "AQ1")
   END_RUNG
   // the same network as SCL:
   "电机启停运行及速度控制"(电机启动 := "电机1启动信号",
                 电机停止 := "电机1停止信号",
                 设定运行时间 := "电机启停运行及速度控制_DB".电机[1].设定运行时间,
                 频率加 := "电机1频率加信号",
                 频率减 := "电机1频率减信号",
                 运行标志 := "电机启停运行及速度控制_DB".电机[1].运行标志,
                 运行时间到 := "电机启停运行及速度控制_DB".电机[1].运行时间到,
                 TON_DB := "电机启停运行及速度控制_DB".电机[1].TON_DB,
                 频率加信号上次状态 := "电机启停运行及速度控制_DB".电机[1].频率加信号上次状态,
                 频率减信号上次状态 := "电机启停运行及速度控制_DB".电机[1].频率减信号上次状态,
                 给定频率 := "电机启停运行及速度控制_DB".电机[1].给定频率,
                 电机输出运行 => "电机1运行",
                 运行指示灯 => "电机1运行指示灯",
                 输出数字量 => "AQ1");
END_REGION

REGION Network 3
   RUNG wire#powerrail
      "电机启停运行及速度控制_FB_DB"(电机启动 :=, 电机停止 :=, 设定运行时间 :=, 频率加 :=, 频率减 :=, 给定频率 :=, 输出数字量 :=, 电机输出运行 =>, 运行指示灯 =>)
   END_RUNG
   // the same network as SCL:
   "电机启停运行及速度控制_FB_DB"();   // "电机启停运行及速度控制_FB"
END_REGION

REGION Network 4
   RUNG wire#powerrail
      "MODBUS通讯_DB"(初始化 :=, 正转 :=, 反转 :=, 停止 :=, 频率设定 :=, 输出频率 =>, 输出电流 =>, 输出电压 =>)
   END_RUNG
   // the same network as SCL:
   "MODBUS通讯_DB"();   // "MODBUS通讯"
END_REGION
END_ORGANIZATION_BLOCK